TYPE ST_ActuatorStatus :
STRUCT
	bEnabled    : BOOL;
    bBusy       : BOOL;
    bDone       : BOOL;
    bError      : BOOL;
    iErrorCode  : UDINT;
    fPosition   : LREAL;
    eState      : E_ActuatorState;
    sMessage    : STRING[80];	
END_STRUCT
END_TYPE

(* stored: Version 1.1.0.1, ProductVersion 3.1.4024.12
   DUT ST_ActuatorStatus: Id {03e2123d-6ce6-49e6-a820-1996bf946a02} *)
